KUKA KRL program: app1b.src, app1b.dat

--- app1b.src ---
&ACCESS RVP
&REL 1
&PARAM DISKPATH = KRC:\R1\Program\arash
DEF app1b( )
;Created by Dumitru Loghin  23_11_2016
;loghindumitru82@gmail.com
;NanoRobotics Laboratory Polytechnique Montreal
;FOLD Declaration
INT i
DECL EKI_STATUS RET
$FLAG[1]=FALSE

;ENDFOLD
;FOLD INI;%{PE}
  ;FOLD BASISTECH INI
    GLOBAL INTERRUPT DECL 3 WHEN $STOPMESS==TRUE DO IR_STOPM ( )
    INTERRUPT ON 3
    BAS (#INITMOV,0 )
  ;ENDFOLD (BASISTECH INI)
  ;FOLD USER INI
    ;Make your modifications here

  ;ENDFOLD (USER INI)
;ENDFOLD (INI)


;FOLD PTP P2 Vel=100 % PDAT2 Tool[1]:Table Base[0];%{PE}%R 8.3.40,%MKUKATPBASIS,%CMOVE,%VPTP,%P 1:PTP, 2:P2, 3:, 5:100, 7:PDAT2
$BWDSTART=FALSE
PDAT_ACT=PPDAT2
FDAT_ACT=FP2
BAS(#PTP_PARAMS,100)
PTP XP2
;ENDFOLD

;FOLD Define callback
INTERRUPT DECL 89 WHEN $FLAG[998]==TRUE DO GET_DATA()
INTERRUPT ON 89
;ENDFOLD

;FOLD ; TTT;%{PE}%R 8.3.40,%MKUKATPBASIS,%CCOMMENT,%VNORMAL,%P 2:TTT
;ENDFOLD
RET=EKI_Init("ConfigApp1")
RET=EKI_Open("ConfigApp1")
WHILE TRUE
;FOLD Write data to connection
; Write frame to <LastPos X="" Y="" Z="" A="" B="" C="" />
RET=EKI_SetFrame("ConfigApp1","Robot/Data/LastPos", $POS_ACT)
; Write int to <Status></Status>
RET=EKI_SetInt("ConfigApp1","Robot/Status", 12345678)
;ENDFOLD
RET = EKI_Send("ConfigApp1","Robot")

$FLAG[1]=FALSE

;wait until data read
WAIT FOR $FLAG[1]

PTP_REL newP
ENDWHILE
RET=EKI_Close("ConfigApp1")
RET=EKI_Clear("ConfigApp1")
END

DEF GET_DATA()
;FOLD Declaration
INT i
DECL EKI_STATUS RET
FRAME valF

;ENDFOLD
;FOLD Initialize sample data
valF={X 0.0,Y 0.0,Z 0.0,A 0.0,B 0.0,C 0.0}

;ENDFOLD
;FOLD Get received sensor data

RET=EKI_GetFrame("ConfigApp1","Pc/Data/SetPos",valF)

newP.x=valF.X
newP.y=valF.Y
newP.z=valF.Z
newP.a=valF.A
newP.b=valF.B
newP.c=valF.C

;ENDFOLD
;FOLD Signal read

$FLAG[998]=FALSE
$FLAG[1]=TRUE

END

--- app1b.dat ---
&ACCESS RVP
&REL 1
&PARAM DISKPATH = KRC:\R1\Program\arash
DEFDAT  app1b PUBLIC
;FOLD EXTERNAL DECLARATIONS;%{PE}%MKUKATPBASIS,%CEXT,%VCOMMON,%P
;FOLD BASISTECH EXT;%{PE}%MKUKATPBASIS,%CEXT,%VEXT,%P
EXT  BAS (BAS_COMMAND  :IN,REAL  :IN )
DECL INT SUCCESS
;ENDFOLD (BASISTECH EXT)
;FOLD USER EXT;%{E}%MKUKATPUSER,%CEXT,%VEXT,%P
;Make your modifications here

;ENDFOLD (USER EXT)
;ENDFOLD (EXTERNAL DECLARATIONS)
DECL E6POS XP1={X 1790.17896,Y -541.692932,Z 1424.40015,A -29.0838795,B -6.69078207,C 0.393054754,S 6,T 18,E1 0.0,E2 0.0,E3 0.0,E4 0.0,E5 0.0,E6 0.0}
DECL BASIS_SUGG_T LAST_BASIS={POINT1[] "P2                      ",POINT2[] "P2                      ",CP_PARAMS[] "CPDAT0                  ",PTP_PARAMS[] "PDAT2                   ",CONT[] "                        ",CP_VEL[] "2.0                     ",PTP_VEL[] "100                     ",SYNC_PARAMS[] "SYNCDAT                 ",SPL_NAME[] "S0                      ",A_PARAMS[] "ADAT0                   "}
DECL FDAT FP1={TOOL_NO 1,BASE_NO 0,IPO_FRAME #BASE,POINT2[] " ",TQ_STATE FALSE}
DECL PDAT PPDAT1={VEL 100.000,ACC 100.000,APO_DIST 100.000,GEAR_JERK 50.0000,EXAX_IGN 0}
DECL GLOBAL POS newP={X -400.000,Y -400.000,Z -400.000,A 0.0,B 0.0,C 0.0}
DECL E6POS XP2={X 1459.79102,Y -1036.28552,Z 919.323547,A -89.4153519,B -1.02977669,C -0.161234230,S 6,T 18,E1 0.0,E2 0.0,E3 0.0,E4 0.0,E5 0.0,E6 0.0}
DECL FDAT FP2={TOOL_NO 1,BASE_NO 0,IPO_FRAME #BASE,POINT2[] " ",TQ_STATE FALSE}
DECL PDAT PPDAT2={VEL 100.000,ACC 100.000,APO_DIST 100.000,GEAR_JERK 50.0000,EXAX_IGN 0}
ENDDAT
